(* CODESYS project Buffer Station - Moraes e Castrucci v2.0_RECOVERED_2026-05-20T00-09-14.project

Project tree, tasks and I/O mapping:
  Device : CODESYS Control Win V3, 3S - Smart Software Solutions GmbH, order no. 305021, version 3.5.11.30
    application Application
      libraries: Standard, * (System)
      task MainTask (cyclic, interval t#20ms, priority 1) calls PLC_PRG
      program PLC_PRG [LD]
      Symbols
*)

// Device/Application/PLC_PRG
PROGRAM PLC_PRG
VAR
	// --- Entradas (Mapear na image_6cef05.png) ---
	aux1				: BOOL; 
	FirstScan			: BOOL;
	xStart_Button       : BOOL; 
	xStop_Button        : BOOL; // NF
	xReset_Button       : BOOL; 
	P0_Home				: BOOL;
	P1_Alimentacao		:BOOL;
	P2_Metal			:BOOL;
	
	
	S_Capacitivo		:BOOL;
	S_Indutivo			:BOOL;
	S_T4_Metal_Out: BOOL;
	S_T3_Plastico_Out: BOOL;

	
END_VAR
VAR // added by the converter: edge detectors and wires of the graphical bodies
    _w1, _w2, _w3, _w4 : BOOL;
    _ft1 : F_TRIG;
    _rt1, _rt2 : R_TRIG;
END_VAR

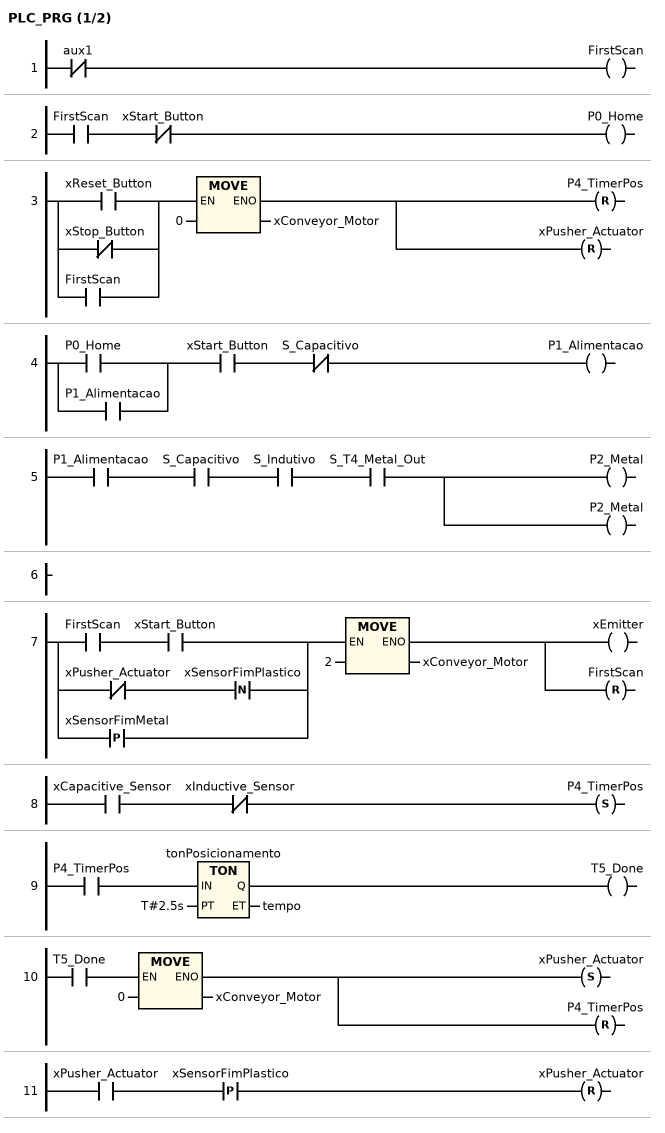
// NETWORK 1
FirstScan := NOT aux1;

// NETWORK 2
P0_Home := FirstScan AND NOT xStart_Button;

// NETWORK 3
_w1 := xReset_Button OR NOT xStop_Button OR FirstScan;
IF _w1 THEN xConveyor_Motor := 0; END_IF
P4_TimerPos R= _w1;
xPusher_Actuator R= _w1;

// NETWORK 4
P1_Alimentacao := (P0_Home OR P1_Alimentacao) AND xStart_Button AND NOT S_Capacitivo;

// NETWORK 5
_w2 := P1_Alimentacao AND S_Capacitivo AND S_Indutivo AND S_T4_Metal_Out;
P2_Metal := _w2;
P2_Metal := _w2;

// NETWORK 6

// NETWORK 7
_ft1(CLK := xSensorFimPlastico);
_rt1(CLK := xSensorFimMetal);
_w3 := FirstScan AND xStart_Button OR NOT xPusher_Actuator AND _ft1.Q OR _rt1.Q;
IF _w3 THEN xConveyor_Motor := 2; END_IF
xEmitter := _w3;
FirstScan R= _w3;

// NETWORK 8
P4_TimerPos S= xCapacitive_Sensor AND NOT xInductive_Sensor;

// NETWORK 9
tonPosicionamento(IN := P4_TimerPos, PT := T#2.5s, ET => tempo); // TON
T5_Done := tonPosicionamento.Q;

// NETWORK 10
_w4 := T5_Done;
IF _w4 THEN xConveyor_Motor := 0; END_IF
xPusher_Actuator S= _w4;
P4_TimerPos R= _w4;

// NETWORK 11
_rt2(CLK := xSensorFimPlastico);
xPusher_Actuator R= xPusher_Actuator AND _rt2.Q;

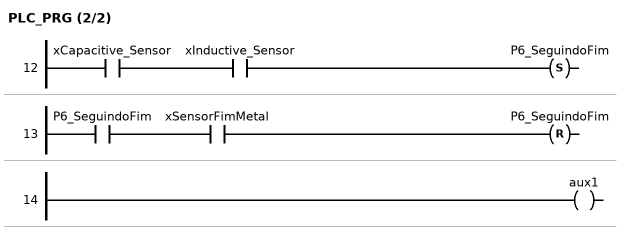
// NETWORK 12
P6_SeguindoFim S= xCapacitive_Sensor AND xInductive_Sensor;

// NETWORK 13
P6_SeguindoFim R= P6_SeguindoFim AND xSensorFimMetal;

// NETWORK 14
aux1 := TRUE;

END_PROGRAM
